{attribute 'GeneratedUsingTerminal: AMP8000-0030-0103-0103'}
{attribute addProperty BoxType "AMP8000-0030-0103-0103"}
{attribute addProperty Id "EtcSlaveTerminalBaseDeviceDevice_6E2575772Device_SafetyDevice_Safety_C21945A160Ch_ACh_A_D18C6F1622WcStateAT %I*WcState_B516A2644InfoDataAT %I*InfoData_358A59CF25"}
{attribute addProperty CRC "2085819216"}
{attribute addProperty Size "113"}
TYPE AMP8000_7C531350 EXTENDS EtcSlaveTerminalBase :
STRUCT
	{attribute addProperty Name "Device"}
	Device : Device_6E257577;
	{attribute addProperty Name "Device_Safety"}
	Device_Safety : Device_Safety_C21945A1;
	{attribute addProperty Name "Ch_A"}
	Ch_A : Ch_A_D18C6F16;
	{attribute addProperty Name "WcState"}
	WcState : WcState_B516A264;
	{attribute addProperty Name "InfoData"}
	InfoData : InfoData_358A59CF;
END_STRUCT
END_TYPE

(* stored: Version 1.2.0.0, ProductVersion 3.1.4024.9
   DUT AMP8000_7C531350: Id {b11ebc80-6656-4b0d-a0e2-b8fc7d392907} *)
